TYPE ST_HMI_PowerMeasDC :
STRUCT
	Voltage : REAL;
	Current	: REAL;
	Power	: REAL;
	SOC		: REAL;
END_STRUCT
END_TYPE

(* stored: Version 1.1.0.1, ProductVersion 3.1.4026.18
   DUT ST_HMI_PowerMeasDC: Id {2dfdd240-99e0-4b6c-b337-99196236d4ca} *)
